METHOD findSearchResults
VAR_INPUT
END_VAR
VAR
	i : INT;
	j : INT;
	searchResult : ST_SearchResult;
END_VAR
FOR i:=0 TO stDoorTrack.CandidateRoutes.CandidateRoutesCount - 1 DO
	FOR j:=0 TO stDoorTrack.CandidateRoutes.CandidateRoutes[i].PathsInfoCount - 1 DO
		searchResult := stSearchResultDefault;
		searchResult.PathIno := stDoorTrack.CandidateRoutes.CandidateRoutes[i].PathsInfo[j];
		searchResult.TargetFeedoutSide := stDoorTrack.CandidateRoutes.CandidateRoutes[i].TargetFeedoutSide;
		addSearchResultToDoorTrack(searchResult);
	END_FOR
END_FOR
END_METHOD

METHOD getFeedMgrStateDescription : STRING
IF config_bIsConveyorTable THEN
	getFeedMgrStateDescription := smC235FeedManager.getStateDescription();
ELSE
	getFeedMgrStateDescription := smC234FeedManager.getStateDescription();
END_IF
END_METHOD

METHOD getSourceAndDestinationIndexFeedoutPortsCount : UINT
IF stDoorTrack.Source < 0 OR stDoorTrack.Source >= MAX_TABLES_COUNT OR
	stDoorTrack.DestinationIndex < 0 OR stDoorTrack.DestinationIndex >= MAX_FEEDOUT_PORTS THEN
	getSourceAndDestinationIndexFeedoutPortsCount := 0;
	RETURN;
END_IF
getSourceAndDestinationIndexFeedoutPortsCount := 
	MAIN.mainStateMachine.smCtrlInterface.
		config_stTransferTableConfig.PrimaryTable.
		Tables[stDoorTrack.Source].DestinationsFeedoutPortsMappingConfig.
		DestinationsFeedoutPortsMappings[stDoorTrack.DestinationIndex].FeedoutPortsCount;
END_METHOD

METHOD getStateDescription : STRING
CASE machineState OF

	TABLEMANAGER_DISABLED:
		getStateDescription := 'Disabled';
			
	TABLEMANAGER_ENABLING:
		getStateDescription := 'Enabling';
			
	TABLEMANAGER_INLINE_JOGGING:
		getStateDescription := 'Inline Jogging';
			
	TABLEMANAGER_CROSS_JOGGING:
		getStateDescription := 'Cross Jogging';
		
	TABLEMANAGER_TO_FENCE_JOGGING:
		getStateDescription := 'To-Fence Jogging';
	
	TABLEMANAGER_ROTATE:
		getStateDescription := 'Rotating';
			
	TABLEMANAGER_SELF_CENTER:
		getStateDescription := 'Centering';
			
	TABLEMANAGER_AUTOFEED_OFF:
		getStateDescription := 'Autofeed Off';
			
	TABLEMANAGER_AUTOFEED_ON:
		getStateDescription := 'Autofeed On';
		
	TABLEMANAGER_DOOR_TRACKER_START:
		getStateDescription := 'Door Track Starting';
			
	TABLEMANAGER_DOOR_TRACKER_WAIT_FOR_DATA_READY_OR_TRANSFERRED_IN:
		IF config_bCanFeedinFromSideA THEN
			getStateDescription := 'Waiting for Door Data Ready or Transferred In';
		ELSE
			getStateDescription := 'Waiting for Door Transferred In';
		END_IF
		
	TABLEMANAGER_DOOR_TRACKER_TRANSFERRING_IN:
		getStateDescription := 'Transferring In';
			
	TABLEMANAGER_DOOR_TRACKER_ROUTE_READY_WAIT_FOR_FEED_IN:
		getStateDescription := 'Route Ready - Waiting for Feed In';
			
	TABLEMANAGER_DOOR_TRACKER_DOOR_FEEDING_IN:
		getStateDescription := 'Door Feeding In';
		
	TABLEMANAGER_DOOR_TRACKER_DOOR_IN_MACHINE_IDLE:
		getStateDescription := 'Door in Machine - Waiting for Transferred Out';

	TABLEMANAGER_DOOR_TRACKER_WAIT_FOR_FEED_OUT:
		IF cmd_bDoorDataReadyLatched THEN
			getStateDescription := 'Waiting for Feed Out. Data Ready Latch Active';
		ELSE
			getStateDescription := 'Waiting for Feed Out';
		END_IF
		
			
	TABLEMANAGER_DOOR_TRACKER_DOOR_FEEDING_OUT:
		getStateDescription := 'Feeding Out';
		
	TABLEMANAGER_DOOR_TRACKER_WAIT_ALL_TABLES_READY:
		getStateDescription := 'Waiting for All Tables Ready';
		
	TABLEMANAGER_DOOR_TRACKER_TRANSFERRING_OUT:
		getStateDescription := 'Transferring Out';
			
	TABLEMANAGER_DOOR_TRACKER_COMPLETE:
		getStateDescription := 'Completed';			
		
	TABLEMANAGER_DOOR_TRACKER_FINDPATH_INIT:
		getStateDescription := 'Finding Path Init';
	
	TABLEMANAGER_DOOR_TRACKER_FINDPATH_RESET:
		getStateDescription := 'Resetting Door Tracker';
		
	TABLEMANAGER_DOOR_TRACKER_FINDPATH_FIND_ENABLED_FEEDOUT_PORTS:
		getStateDescription := 'Finding Enabled Feedout Ports';
		
	TABLEMANAGER_DOOR_TRACKER_FINDPATH_WAITING_FOR_CLEAR_ROUTE:
		getStateDescription := 'Waiting for Clear Route';
	
	TABLEMANAGER_DOOR_TRACKER_FINDPATH_FIND_CANDIDATE_ROUTES:
		getStateDescription := 'Finding Candidate Routes';
		
	TABLEMANAGER_DOOR_TRACKER_FINDPATH_FIND_SEARCH_RESULTS:
		getStateDescription := 'Finding Search Results';
		
	TABLEMANAGER_DOOR_TRACKER_FINDPATH_COMPUTE_FINAL_SCORE:
		getStateDescription := 'Computing Final Score';
		
	TABLEMANAGER_DOOR_TRACKER_FINDPATH_REQUEST_NEW_ROUTE_COMPLETE:
		getStateDescription := 'Request New Route Complete';
		
	TABLEMANAGER_DOOR_TRACKER_FINDPATH_COMPLETE:
		getStateDescription := 'Finding Path Complete';
	
	TABLEMANAGER_DOOR_TRACKER_ALL_TARGET_FEEDOUT_PORTS_DISABLED:
		getStateDescription := 'All of Target Feed-out Ports Disabled';	

	TABLEMANAGER_DOOR_TRACKER_DOOR_HAS_NO_TARGET:
		getStateDescription := 'Door Has No Target';
		
	TABLEMANAGER_ERROR:
		getStateDescription := 'Error';
		
END_CASE
END_METHOD

METHOD getTargetNodeDirection : E_Direction
VAR 
	i : INT;
END_VAR
getTargetNodeDirection := E_Direction.None;
IF NOT bHasDoor THEN
	RETURN;
END_IF

FOR i:= 0 TO stDoorTrack.TargetPath.PathCount - 1 DO
	// do we have the source from TargetPath?
	IF stDoorTrack.TargetPath.Path[i].TableIndex = config_iTableArrayIndex THEN
		getTargetNodeDirection := stDoorTrack.TargetPath.Path[i].Direction;
		RETURN;
	END_IF
END_FOR
END_METHOD

METHOD goFast
VAR_INPUT
END_VAR
psmHcFeedMotor^.cmd_bSpeedFast := TRUE;
END_METHOD

METHOD goFwd
VAR_INPUT
END_VAR
psmHcFeedMotor^.cmd_bFwd := TRUE;
END_METHOD

METHOD goRev
VAR_INPUT
END_VAR
psmHcFeedMotor^.cmd_bRev := TRUE;
END_METHOD

METHOD goSlow
VAR_INPUT
END_VAR
psmHcFeedMotor^.cmd_bSpeedSlow := TRUE;
END_METHOD

METHOD hasDeadlockedDoorInPath : BOOL
VAR_INPUT
	pstPath : POINTER TO ST_PathInfo;
END_VAR
VAR
	i : INT;
END_VAR
hasDeadlockedDoorInPath := FALSE;
IF pstPath = 0 THEN	
	RETURN;
END_IF

FOR i:= 0 TO pstPath^.PathCount - 1 DO
	IF MAIN.mainStateMachine.asmTableManagers[pstPath^.Path[i].TableIndex].bHasDoor AND 
		(MAIN.mainStateMachine.asmTableManagers[pstPath^.Path[i].TableIndex].bWaitingForClearRoute OR
		MAIN.mainStateMachine.asmTableManagers[pstPath^.Path[i].TableIndex].bAllTargetFeedoutPortsDisabled OR
		MAIN.mainStateMachine.asmTableManagers[pstPath^.Path[i].TableIndex].bDoorHasNoTarget)
	THEN
		hasDeadlockedDoorInPath := TRUE;
		RETURN;
	END_IF
END_FOR
END_METHOD

METHOD hasDoorGoingOppositeDirection : BOOL
VAR_INPUT
	pstPath : POINTER TO ST_PathInfo;
END_VAR
VAR
	i : INT;
	j : INT;
	k : INT;
	intersectAtTableIndex : INT;
	prevDoorDirection : E_Direction;
	curDoorDirection : E_Direction;
	otherDoorDirection : E_Direction;
	pstPathOther : POINTER TO ST_PathInfo;
END_VAR
hasDoorGoingOppositeDirection := FALSE;
IF pstPath = 0 THEN	
	RETURN;
END_IF

FOR i:= 0 TO pstPath^.PathCount - 1 DO
	intersectAtTableIndex := pstPath^.Path[i].TableIndex;
	IF MAIN.mainStateMachine.asmTableManagers[intersectAtTableIndex].stDoorTrack.Target <> -1 THEN
		pstPathOther := ADR(MAIN.mainStateMachine.asmTableManagers[intersectAtTableIndex].stDoorTrack.TargetPath);
		FOR j:= 0 TO pstPathOther^.PathCount - 1 DO
			prevDoorDirection := E_Direction.None;
			FOR k:= 0 TO pstPath^.PathCount - 1 DO				
				curDoorDirection := pstPath^.Path[k].Direction;
				IF pstPathOther^.Path[j].TableIndex = pstPath^.Path[k].TableIndex THEN
					otherDoorDirection  := pstPathOther^.Path[j].Direction;
					IF 	curDoorDirection = E_Direction.North 	AND otherDoorDirection = E_Direction.South OR
						curDoorDirection = E_Direction.South 	AND otherDoorDirection = E_Direction.North OR
						curDoorDirection = E_Direction.West 	AND otherDoorDirection = E_Direction.East OR
						curDoorDirection = E_Direction.East 	AND otherDoorDirection = E_Direction.West OR
						prevDoorDirection = E_Direction.North 	AND otherDoorDirection = E_Direction.South OR
						prevDoorDirection = E_Direction.South 	AND otherDoorDirection = E_Direction.North OR
						prevDoorDirection = E_Direction.West 	AND otherDoorDirection = E_Direction.East OR
						prevDoorDirection = E_Direction.East 	AND otherDoorDirection = E_Direction.West
					THEN
						hasDoorGoingOppositeDirection := TRUE;
						RETURN;
					END_IF
				END_IF
				prevDoorDirection := curDoorDirection;
			END_FOR
		END_FOR
	END_IF
END_FOR
END_METHOD

METHOD hasEmptyTableInPath : BOOL
VAR_INPUT
	pstPath : POINTER TO ST_PathInfo;
END_VAR
VAR
	i : INT;
END_VAR
IF pstPath = 0 THEN
	hasEmptyTableInPath := FALSE;
	RETURN;
END_IF

IF pstPath^.PathCount = 0 THEN
	hasEmptyTableInPath := FALSE;
	RETURN;
END_IF

IF pstPath^.PathCount = 1 THEN
	hasEmptyTableInPath := NOT MAIN.mainStateMachine.asmTableManagers[pstPath^.Path[0].TableIndex].bHasDoor;
	RETURN;
END_IF

// skip index 0, which is the source/first table in path.
FOR i:= 1 TO pstPath^.PathCount - 1 DO
	IF NOT MAIN.mainStateMachine.asmTableManagers[pstPath^.Path[i].TableIndex].bHasDoor THEN
		hasEmptyTableInPath := TRUE;
		RETURN;
	END_IF
END_FOR

hasEmptyTableInPath := FALSE;
END_METHOD

METHOD hasError : bool
hasError := smDoorDasher.bError;
IF hasError THEN
	RETURN;
END_IF

IF config_bIsConveyorTable THEN
	hasError := smC235FeedManager.bError;
ELSE
	hasError := smC234FeedManager.bError;
END_IF
END_METHOD

METHOD hasErrorDescription : T_MaxString
hasErrorDescription := smDoorDasher.sError;
IF hasErrorDescription <> '' THEN
	RETURN;
END_IF

IF config_bIsConveyorTable THEN
	hasErrorDescription := smC235FeedManager.sError;
ELSE
	hasErrorDescription := smC234FeedManager.sError;
END_IF
END_METHOD

METHOD hasErrorId : UINT
hasErrorId := INT_TO_UINT(smDoorDasher.iLastErrorId);
IF hasErrorId <> 0 THEN
	RETURN;
END_IF

IF config_bIsConveyorTable THEN
	hasErrorId := INT_TO_UINT(smC235FeedManager.iLastErrorId);
ELSE
	hasErrorId := INT_TO_UINT(smC234FeedManager.iLastErrorId);
END_IF
END_METHOD

METHOD hasIncomingDoorInPath : BOOL
VAR_INPUT
	pstPath : POINTER TO ST_PathInfo;
END_VAR
VAR
	i : INT;
END_VAR
hasIncomingDoorInPath := FALSE;
IF pstPath = 0 THEN	
	RETURN;
END_IF

FOR i:= 0 TO pstPath^.PathCount - 1 DO
	IF MAIN.mainStateMachine.asmTableManagers[pstPath^.Path[i].TableIndex].bRouteReadyWaitForFeedIn THEN
		hasIncomingDoorInPath := TRUE;
		RETURN;
	END_IF
END_FOR
END_METHOD

METHOD initDoorTrack
VAR_INPUT
END_VAR
stDoorTrackLast := stDoorTrack; 

stDoorTrack.CandidateRoutes := stCandidateRoutesDefault;
stDoorTrack.SearchResults := stSearchResultsDefault;
stDoorTrack.TargetPath := stPathInfoDefault;

bHasEnabledFeedoutPorts := FALSE;

IF cmd_bRequestNewRoute THEN
	stDoorTrack.AllEnabledFeedoutPorts := stFeedoutPortsConfigDefault;
	stDoorTrack.RejectedFeedoutPorts := stFeedoutPortsConfigDefault;
	stDoorTrack.ReroutableFeedoutPorts := stReroutableFeedoutPortsConfigDefault;
	stDoorTrack.RejectedFeedoutPorts.FeedoutPortsCount := -1; // Notifies HMI to clear the rejected feed-out ports list for operator's manual re-route.
	stDoorTrack.ReroutableFeedoutPorts.FeedoutPortsCount := -1; // Notifies HMI to clear the reroutable feed-out ports list for operator's manual re-route.
ELSE
	stDoorTrack.TargetFeedoutPorts := stFeedoutPortsConfigDefault;
	stDoorTrack.DoorIsRotating := FALSE;
	stDoorTrack.DoorRotateRequired := FALSE;
	stDoorTrack.DoorWasRotated := FALSE;
END_IF
END_METHOD

METHOD initialize
VAR CONSTANT		
END_VAR
SUPER^.initialize();

descriptor.sModuleClass := 'TableManager';

// TODO: don't init if config_pstHcTransferTableHardware and config_pstHcConveyorHardware are null
config_pstHcTransferTableHardware;
config_pstHcConveyorHardware;

// initialize machine configs and defaults
cmd_bManualControlEnabled := config_bManualControlEnabled;

(*     --- Feed System ---     *)
IF config_bIsConveyorTable THEN
	//
	iCrossFeedFastSpeedRpm	:= LREAL_TO_UINT(config_iCrossFeedFastSpeedFPM / CONVEYOR_CROSSFEED_RPM_TO_FPM);
	iCrossFeedSlowSpeedRpm	:= LREAL_TO_UINT(config_iCrossFeedSlowSpeedFPM / CONVEYOR_CROSSFEED_RPM_TO_FPM);
	iFeedFastSpeedRPM		:= iCrossFeedFastSpeedRpm;
	iFeedSlowSpeedRPM 		:= iCrossFeedSlowSpeedRpm;
	iFeedOutSpeedRPM		:= 0; // not used for Conveyor table
	IF (config_pstHcConveyorHardware <> 0) THEN
		psmHcFeedMotor := ADR(config_pstHcConveyorHardware^.smFeedMotor);
	END_IF
ELSE
	//
	iCrossFeedFastSpeedRpm	:= LREAL_TO_UINT(config_iCrossFeedFastSpeedFPM / TABLE_CROSSFEED_RPM_TO_FPM);
	iCrossFeedSlowSpeedRpm	:= LREAL_TO_UINT(config_iCrossFeedSlowSpeedFPM / TABLE_CROSSFEED_RPM_TO_FPM);
	iFeedFastSpeedRPM		:= LREAL_TO_UINT(config_iFeedFastSpeedFPM / TABLE_INLINE_FEED_RPM_TO_FPM);
	iFeedSlowSpeedRPM 		:= LREAL_TO_UINT(config_iFeedSlowSpeedFPM / TABLE_INLINE_FEED_RPM_TO_FPM);
	iFeedOutSpeedRPM		:= LREAL_TO_UINT(config_iFeedOutSpeedFPM  / TABLE_INLINE_FEED_RPM_TO_FPM);
	IF (config_pstHcTransferTableHardware <> 0) THEN
		psmHcFeedMotor := ADR(config_pstHcTransferTableHardware^.smFeedMotor);
	END_IF
END_IF

IF (psmHcFeedMotor = 0) THEN
	logger(ePriority := E_LogPriority.LOGPRIORITY_WARNING_LOW, sMessage := 'Incorrect config - assigning dummy pointer to VFD');
	psmHcFeedMotor := ADR(MAIN.mainStateMachine.smDummyMotor);
END_IF
	
{IF defined (noHW) OR defined (noHW_UML)}
	// these are for no hardware mode only...
	psmHcFeedMotor^.config_bNoHardwareTestMode := config_bNoHardwareTestMode;
	psmHcFeedMotor^.config_fTestMaxAccel := 24; // unit: in/s^2
	psmHcFeedMotor^.config_fTestMaxDecel := 24; // unit: in/s^2
	psmHcFeedMotor^.config_fTestMaxJerk := 144; // unit: in/s^3
	psmHcFeedMotor^.config_fTestMaxSpeed := 30; // unit : in/sec
	
	IF psmHcFeedMotor^.config_iFastSpeedRPM = 0 THEN
		psmHcFeedMotor^.config_iFastSpeedRPM := 1345;
	END_IF
	psmHcFeedMotor^.config_fUnitConversionFactor := (config_iFeedFastSpeedFPM * 12.0) / (psmHcFeedMotor^.config_iFastSpeedRPM * 60.0);
{END_IF}

// Assign dummy values preemptively - if have correct link to hardware, will get overwritten
// Have to assign these here, in initialize, because SM_TableManager references some of these in preProcess
smC234FeedManager.psmCrossFeedFenceHeightCyl 					:= ADR(MAIN.mainStateMachine.smDummyCylinder);
smC234FeedManager.psmCrossFeedTransferHeightCyl 				:= ADR(MAIN.mainStateMachine.smDummyCylinder);
smC234FeedManager.smSelfCenterManager.psmSelfCenterWheelsCyl 	:= ADR(MAIN.mainStateMachine.smDummyCylinder);
smC234FeedManager.smSelfCenterManager.psmSelfCenterCyl 			:= ADR(MAIN.mainStateMachine.smDummyCylinder);
smC234FeedManager.smRotateManager.psmDoorLiftCyl				:= ADR(MAIN.mainStateMachine.smDummyCylinder);
smC234FeedManager.smRotateManager.psmRotateCyl					:= ADR(MAIN.mainStateMachine.smDummyDoubleCylinder);
	
IF config_bIsConveyorTable THEN
	addChildStateMachine('C235 Feed Manager', ADR(smC235FeedManager)); 
		smC235FeedManager.pbTableIsEmpty := ADR(bTableIsEmpty);
		smC235FeedManager.pbDoorInMachine := ADR(bDoorInMachine);
		smC235FeedManager.pstTable := THIS;
		smC235FeedManager.pstDoorTrack := ADR(stDoorTrack);
		smC235FeedManager.itfDoorTracker := THIS^;
		smC235FeedManager.psmFeedMotor := psmHcFeedMotor;
		smC235FeedManager.config_iFeedOutSpeedRPM := iCrossFeedFastSpeedRPM;
		smC235FeedManager.config_iCrossFastSpeedRPM := iCrossFeedFastSpeedRPM;
		smC235FeedManager.config_iCrossSlowSpeedRPM := iCrossFeedSlowSpeedRPM;
		smC235FeedManager.config_bNoHardwareTestMode := config_bNoHardwareTestMode;
		smC235FeedManager.config_iTableArrayIndex := config_iTableArrayIndex;
ELSE		
	addChildStateMachine('C234 Feed Manager', ADR(smC234FeedManager));
		smC234FeedManager.pbTableIsEmpty := ADR(bTableIsEmpty);
		smC234FeedManager.pbDoorInMachine := ADR(bDoorInMachine);
		smC234FeedManager.pstTable := THIS;
		smC234FeedManager.pstDoorTrack := ADR(stDoorTrack);
		smC234FeedManager.itfDoorTracker := THIS^;
		smC234FeedManager.config_bCanRotate := config_bCanRotate;
		smC234FeedManager.config_bCanSelfCenter := config_bCanSelfCenter;
		smC234FeedManager.config_bIsBufferTable := config_bIsBufferTable;
		smC234FeedManager.psmFeedMotor := psmHcFeedMotor;
		smC234FeedManager.config_iFastSpeedRPM := iFeedFastSpeedRPM;
		smC234FeedManager.config_iSlowSpeedRPM := iFeedSlowSpeedRPM;
		smC234FeedManager.config_iFeedOutSpeedRPM := iFeedOutSpeedRPM;
		smC234FeedManager.config_iCrossFastSpeedRPM := iCrossFeedFastSpeedRPM;
		smC234FeedManager.config_iCrossSlowSpeedRPM := iCrossFeedSlowSpeedRPM;
		smC234FeedManager.config_bNoHardwareTestMode := config_bNoHardwareTestMode;
		smC234FeedManager.config_iTableArrayIndex := config_iTableArrayIndex;
		// Assign valve pointers
		IF (config_pstHcTransferTableHardware <> 0) THEN
			smC234FeedManager.psmCrossFeedFenceHeightCyl 					:= ADR(config_pstHcTransferTableHardware^.smCrossFeedFenceHeightCyl);
			smC234FeedManager.psmCrossFeedTransferHeightCyl 				:= ADR(config_pstHcTransferTableHardware^.smCrossFeedTransferHeightCyl);
			smC234FeedManager.smSelfCenterManager.psmSelfCenterWheelsCyl 	:= ADR(config_pstHcTransferTableHardware^.smSelfCenterWheelsCyl);
			smC234FeedManager.smSelfCenterManager.psmSelfCenterCyl 			:= ADR(config_pstHcTransferTableHardware^.smSelfCenterCyl);
			smC234FeedManager.smRotateManager.psmDoorLiftCyl 				:= ADR(config_pstHcTransferTableHardware^.smDoorLiftCyl);
			smC234FeedManager.smRotateManager.psmRotateCyl 					:= ADR(config_pstHcTransferTableHardware^.smRotateCyl);
		ELSE
			logger(ePriority := E_LogPriority.LOGPRIORITY_WARNING_LOW, sMessage := 'Incorrect config - assigning dummy pointer to valves');
		END_IF
END_IF

addChildStateMachine('Door Dasher', ADR(smDoorDasher));
	smDoorDasher(
		pstTable := THIS,
		pstDoorTrack := ADR(stDoorTrack),
		itfDoorTracker := THIS^,
		config_bNoHardwareTestMode := config_bNoHardwareTestMode,
		config_iTableArrayIndex := config_iTableArrayIndex
	);
END_METHOD

METHOD initInputSourceAndDestinationIndexWithHighestFeedoutPortsCount : BOOL
VAR_IN_OUT
	iInputSource	: INT;
	iDestinationIndex	: INT;
END_VAR
VAR 
	iInputSourceIndex : INT;
	iDestIndex : INT;
	feedoutPortsCountMax : INT;
END_VAR
iInputSource := 0;
iDestinationIndex := 0;
feedoutPortsCountMax := 0;

FOR iInputSourceIndex:=0 TO MAIN.mainStateMachine.smCtrlInterface.config_stTransferTableConfig.PrimaryTable.TablesCount-1 DO
	IF NOT (MAIN.mainStateMachine.smCtrlInterface.config_stTransferTableConfig.PrimaryTable.Tables[iInputSourceIndex].IsFunctionalTable AND
			MAIN.mainStateMachine.asmTableManagers[iInputSourceIndex].config_bCanFeedinFromSideA) THEN
		CONTINUE;
	END_IF
	IF MAIN.mainStateMachine.smCtrlInterface.config_stTransferTableConfig.PrimaryTable.Tables[iInputSourceIndex].DestinationsFeedoutPortsMappingConfig.DestinationsFeedoutPortsMappingsCount > 0 THEN
		FOR iDestIndex:=0 TO MAIN.mainStateMachine.smCtrlInterface.config_stTransferTableConfig.PrimaryTable.Tables[iInputSourceIndex].DestinationsFeedoutPortsMappingConfig.DestinationsFeedoutPortsMappingsCount - 1 DO
			IF MAIN.mainStateMachine.smCtrlInterface.config_stTransferTableConfig.PrimaryTable.Tables[iInputSourceIndex].DestinationsFeedoutPortsMappingConfig.DestinationsFeedoutPortsMappings[iDestIndex].FeedoutPortsCount > feedoutPortsCountMax THEN
				iInputSource := iInputSourceIndex;
				iDestinationIndex := MAIN.mainStateMachine.smCtrlInterface.config_stTransferTableConfig.PrimaryTable.Tables[iInputSourceIndex].DestinationsFeedoutPortsMappingConfig.DestinationsFeedoutPortsMappings[iDestIndex].DestinationIndex;
				feedoutPortsCountMax := MAIN.mainStateMachine.smCtrlInterface.config_stTransferTableConfig.PrimaryTable.Tables[iInputSourceIndex].DestinationsFeedoutPortsMappingConfig.DestinationsFeedoutPortsMappings[iDestIndex].FeedoutPortsCount;
			END_IF
		END_FOR
	END_IF
END_FOR
END_METHOD

METHOD isCurrentTargetFeedoutPortEnabled : BOOL
VAR_INPUT
END_VAR
isCurrentTargetFeedoutPortEnabled := FALSE;
IF 	stDoorTrack.Target <> -1 THEN		
	isCurrentTargetFeedoutPortEnabled := MAIN.mainStateMachine.asmTableManagers[stDoorTrack.Target].isFeedoutSideEnabled(stDoorTrack.TargetFeedoutSide);
END_IF
END_METHOD

// if currentTargetFeedoutPort exists in DestinationIndex, then the current Target was a re-route.
METHOD isCurrentTargetFeedoutPortExistInDestinationIndexFeedoutPorts : BOOL
VAR_INPUT
END_VAR
VAR
	i : INT;
	j : INT;
	k : INT;
	stFeedoutPort : ST_FeedoutPort;
END_VAR
isCurrentTargetFeedoutPortExistInDestinationIndexFeedoutPorts := FALSE;
IF 	stDoorTrack.DestinationIndex <> -1 AND
	stDoorTrack.Target <> -1 
	THEN
	i := stDoorTrack.Source;
	IF MAIN.mainStateMachine.smCtrlInterface.config_stTransferTableConfig.PrimaryTable.Tables[i].DestinationsFeedoutPortsMappingConfig.DestinationsFeedoutPortsMappingsCount > 0 THEN
		FOR j:=0 TO MAIN.mainStateMachine.smCtrlInterface.config_stTransferTableConfig.PrimaryTable.Tables[i].DestinationsFeedoutPortsMappingConfig.DestinationsFeedoutPortsMappingsCount - 1 DO
			IF MAIN.mainStateMachine.smCtrlInterface.config_stTransferTableConfig.PrimaryTable.Tables[i].DestinationsFeedoutPortsMappingConfig.DestinationsFeedoutPortsMappings[j].DestinationIndex = stDoorTrack.DestinationIndex THEN
				IF MAIN.mainStateMachine.smCtrlInterface.config_stTransferTableConfig.PrimaryTable.Tables[i].DestinationsFeedoutPortsMappingConfig.DestinationsFeedoutPortsMappings[j].FeedoutPortsCount > 0 THEN
					FOR k:=0 TO MAIN.mainStateMachine.smCtrlInterface.config_stTransferTableConfig.PrimaryTable.Tables[i].DestinationsFeedoutPortsMappingConfig.DestinationsFeedoutPortsMappings[j].FeedoutPortsCount - 1 DO
						stFeedoutPort := MAIN.mainStateMachine.smCtrlInterface.config_stTransferTableConfig.PrimaryTable.Tables[i].DestinationsFeedoutPortsMappingConfig.DestinationsFeedoutPortsMappings[j].FeedoutPorts[k];
						IF stFeedoutPort.TableIndex = stDoorTrack.Target AND stFeedoutPort.Side = stDoorTrack.TargetFeedoutSide THEN
							isCurrentTargetFeedoutPortExistInDestinationIndexFeedoutPorts := TRUE;
							RETURN;
						END_IF
					END_FOR
				END_IF
				EXIT;
			END_IF
		END_FOR
	END_IF
END_IF
END_METHOD

METHOD isFeedoutSideEnabled : BOOL
VAR_INPUT
	eFeedoutSide : E_FeedoutSideType;
END_VAR
isFeedoutSideEnabled := FALSE;
IF config_bIsConveyorTable THEN
	IF eFeedoutSide = E_FeedoutSideType.C THEN
		isFeedoutSideEnabled := NOT smC235FeedManager.di_DisableFeedoutSideC;
	ELSIF eFeedoutSide = E_FeedoutSideType.D THEN
		isFeedoutSideEnabled := NOT smC235FeedManager.di_DisableFeedoutSideD;
	END_IF
ELSE
	IF eFeedoutSide = E_FeedoutSideType.A THEN
		isFeedoutSideEnabled := NOT smC234FeedManager.di_DisableFeedoutSideA;
	ELSIF eFeedoutSide = E_FeedoutSideType.B THEN
		isFeedoutSideEnabled := NOT smC234FeedManager.di_DisableFeedoutSideB;
	ELSIF eFeedoutSide = E_FeedoutSideType.C THEN
		isFeedoutSideEnabled := NOT smC234FeedManager.di_DisableFeedoutSideC;
	ELSIF eFeedoutSide = E_FeedoutSideType.D THEN
		isFeedoutSideEnabled := NOT smC234FeedManager.di_DisableFeedoutSideD;
	END_IF
END_IF
END_METHOD

METHOD isNeighborInTargetPath : BOOL
VAR_INPUT
	neighborIndex : INT;
END_VAR
VAR 
	i : INT;
END_VAR
isNeighborInTargetPath := FALSE;

FOR i:= 0 TO stDoorTrack.TargetPath.PathCount - 1 DO
	// do we have the neighborIndex in TargetPath?
	IF stDoorTrack.TargetPath.Path[i].TableIndex = neighborIndex THEN
		isNeighborInTargetPath := TRUE;
		RETURN;
	END_IF
END_FOR
END_METHOD

METHOD isTableIndexExistInCandidateRoutes : BOOL
VAR_INPUT
	iTableIndex : INT;
END_VAR
VAR
	i : INT;
END_VAR
isTableIndexExistInCandidateRoutes := FALSE;
FOR i:=0 TO stDoorTrack.CandidateRoutes.CandidateRoutesCount-1 DO
	IF stDoorTrack.CandidateRoutes.CandidateRoutes[i].TargetTableIndex = iTableIndex THEN
		isTableIndexExistInCandidateRoutes := TRUE;
		RETURN;
	END_IF
END_FOR
END_METHOD

METHOD minDirectionalChanges : LREAL
VAR_INPUT
	pstSearchResults : POINTER TO ST_SearchResults;
END_VAR
VAR
	i : INT;
	pstSearchResult : POINTER TO ST_SearchResult;
	minDirChanges : LREAL := MAX_LREAL;
END_VAR
IF pstSearchResults = 0 THEN
	RETURN;
END_IF

FOR i:=0 TO pstSearchResults^.SearchResultsCount - 1 DO
	pstSearchResult := ADR(pstSearchResults^.SearchResults[i]);
	IF pstSearchResult^.DirectionalChanges < minDirChanges THEN
		minDirChanges := pstSearchResult^.DirectionalChanges;
	END_IF
END_FOR

minDirectionalChanges := minDirChanges;
END_METHOD

METHOD minDoorsInPath : LREAL
VAR_INPUT
	pstSearchResults : POINTER TO ST_SearchResults;
END_VAR
VAR
	i : INT;
	pstSearchResult : POINTER TO ST_SearchResult;
	minDoorIntersects : LREAL := MAX_LREAL;
END_VAR
IF pstSearchResults = 0 THEN
	RETURN;
END_IF

FOR i:=0 TO pstSearchResults^.SearchResultsCount - 1 DO
	pstSearchResult := ADR(pstSearchResults^.SearchResults[i]);
	IF pstSearchResult^.DoorsInPath < minDoorIntersects THEN
		minDoorIntersects := pstSearchResult^.DoorsInPath;
	END_IF
END_FOR

minDoorsInPath := minDoorIntersects;
END_METHOD

METHOD minNumberOfHops : LREAL
VAR_INPUT
	pstSearchResults : POINTER TO ST_SearchResults;
END_VAR
VAR
	i : INT;
	pstSearchResult : POINTER TO ST_SearchResult;
	minHops : LREAL := MAX_LREAL;
END_VAR
IF pstSearchResults = 0 THEN
	RETURN;
END_IF

FOR i:=0 TO pstSearchResults^.SearchResultsCount - 1 DO
	pstSearchResult := ADR(pstSearchResults^.SearchResults[i]);
	IF pstSearchResult^.NumberOfHops < minHops THEN
		minHops := pstSearchResult^.NumberOfHops;
	END_IF
END_FOR

minNumberOfHops := minHops;
END_METHOD

METHOD pathHasRotateOption : BOOL
VAR_INPUT
	pstPath : POINTER TO ST_PathInfo;
END_VAR
VAR
	i : INT;
	nodeTableIndex : INT;
END_VAR
pathHasRotateOption := FALSE;
IF pstPath = 0 THEN	
	RETURN;
END_IF

FOR i:= 0 TO pstPath^.PathCount - 1 DO
	nodeTableIndex := pstPath^.Path[i].TableIndex;
	IF MAIN.mainStateMachine.asmTableManagers[nodeTableIndex].config_bCanRotate THEN
		pathHasRotateOption := TRUE;
		RETURN;
	END_IF
END_FOR
END_METHOD

METHOD postProcess
VAR_INPUT
END_VAR
SUPER^.postProcess();
cmd_bAbort := FALSE;
cmd_bRotate			:= FALSE;
cmd_bSelfCenter			:= FALSE;	
cmd_bExternal		:= FALSE;	
cmd_bInternal			:= FALSE;	
cmd_bFeedinStarted	:= FALSE;
cmd_bFeedinCompleted := FALSE;
cmd_bFeedoutStarted := FALSE;
cmd_bFeedoutCompleted := FALSE;
cmd_bDoorTransferInStarted := FALSE;
cmd_bDoorTransferInCompleted := FALSE;
cmd_bDoorTransferOutCompleted := FALSE;
END_METHOD

(* this method is run before the doState is run*)
METHOD preProcess
SUPER^.preProcess();

// Jamb kickover
IF (config_pstHcTransferTableHardware <> 0) THEN
	tofJambKickOverTimer(IN:=config_bCanFeedinFromSideA AND config_pstHcTransferTableHardware^.di_JambKickoverEye, PT:=T#2.0S);
	config_pstHcTransferTableHardware^.do_jambKickover := tofJambKickOverTimer.Q AND (NOT config_pstHcTransferTableHardware^.di_JambKickoverEye);
END_IF

// persist configs to disk
rtrigPersistentDataChanged(CLK:=
	config_bManualControlEnabled <> cmd_bManualControlEnabled);
IF rtrigPersistentDataChanged.Q THEN
	config_bManualControlEnabled := cmd_bManualControlEnabled;
END_IF
bExternal := anyChildExternal();
status_bBusy := anyChildBusy() OR smDoorDasher.status_bBusy;
status_bMoving := psmHcFeedMotor^.status_bMoving;
bReadyToRotate := 
	NOT (smC234FeedManager.smRotateManager.psmDoorLiftCyl^.status_bFloating OR smC234FeedManager.smRotateManager.psmRotateCyl^.status_bFloating) AND
	(smC234FeedManager.smSelfCenterManager.psmSelfCenterCyl^.status_bRetracted OR NOT config_bCanSelfCenter);
bOkToSelfCenter := smC234FeedManager.smRotateManager.bDoorLiftCylRetracted OR NOT config_bCanRotate;

bHasDoor := bDoorInMachine;
ftrigHasDoor(CLK:=bHasDoor);

rtrigAutofeedOn(CLK:=cmd_bAutoFeedOn);
IF rtrigAutofeedOn.Q THEN
	autofeedOn();
END_IF

// Eye blowoff
IF (config_pstHcTransferTableHardware <> 0) THEN
	IF rtrigAutofeedOn.Q OR ftrigHasDoor.Q THEN
		config_pstHcTransferTableHardware^.do_eyeBlowoff := TRUE;
	END_IF
	tonEyeBlowoffTimer(IN:=config_pstHcTransferTableHardware^.do_eyeBlowoff, PT:=T#1S);
	IF tonEyeBlowoffTimer.Q THEN
		config_pstHcTransferTableHardware^.do_eyeBlowoff := FALSE;
	END_IF
END_IF

ftrigAnyChildNotAutofeedOn(CLK:=allChildrenAutoFeedOn());
IF ftrigAnyChildNotAutofeedOn.Q THEN
	cmd_bAutoFeedOn := FALSE;
END_IF

ftrigAutofeedOn(CLK:=cmd_bAutoFeedOn);
IF ftrigAutofeedOn.Q THEN
	autofeedOff();
END_IF


rtrigExternal(CLK:=cmd_bExternal);
IF rtrigExternal.Q THEN
	setExternal();
END_IF

rtrigExternal(CLK:=cmd_bInternal);
IF rtrigExternal.Q THEN
	setInternal();
END_IF

rtrigTableIndexNotExistInDoorTrackTargetPath(CLK:= 
	bHasDoor AND 
	stDoorTrack.Target <> -1 AND 
	stDoorTrack.TargetPath.PathCount > 0 AND 
	NOT existTableIndexInDoorTrackTargetPath());

rtrigRequestNewRoute(CLK:=cmd_bRequestNewRoute);

// cmd_bIncomingDoorHandValid := di_IncomingDoorLH XOR di_IncomingDoorRH
cmd_bIncomingDoorHandValid := cmd_eIncomingDoorHand <> E_DOORHAND.DOORHAND_NO_HAND;

// Monitor cmd_bIncomingDoorHandValid on falling edge. The feeding machine (ie, 994-X) clears LH/RH inputs on completion of its feed-out seq. 
ftrigIncomingDoorHandValid(CLK:=cmd_bIncomingDoorHandValid);

// Monitor on rising edge. The feeding machine (ie, 994-X) sets LH/RH inputs at start of its feed-out seq. 
rtrigIncomingDoorHandChanged(CLK:=cmd_bIncomingDoorHandValid AND cmd_eIncomingDoorHandLast <> cmd_eIncomingDoorHand);

cmd_eIncomingDoorHandLast := cmd_eIncomingDoorHand;

bSelectedDestinationIndexChanged := cmd_iSelectedDestinationIndexLast <> cmd_iSelectedDestinationIndex;
cmd_iSelectedDestinationIndexLast := cmd_iSelectedDestinationIndex;


bAutoDataReadyConfigChanged := bAutoDataReadyConfigLast <> config_bAutoDataReady;
bAutoDataReadyConfigLast := config_bAutoDataReady;

rtrigAutoDataReadyChanged(clk:=bAutoDataReadyConfigChanged);

IF bSelectedDestinationIndexChanged OR bAutoDataReadyConfigChanged THEN
	setDoorDataReadyLatch(FALSE);
END_IF

tofSelectedDestinationIndexChangedTimer(IN := bSelectedDestinationIndexChanged, PT := T#100MS);

// Detect falling edge of the input signal
ftrigSelectedDestinationIndexChanged(CLK := tofSelectedDestinationIndexChangedTimer.Q);

IF ftrigSelectedDestinationIndexChanged.Q THEN	
	bAnySourceDestinationIndexFeedoutPortEnabled := anySourceDestinationIndexFeedoutPortEnabled(UINT_TO_INT(cmd_iSelectedDestinationIndex));
	cmd_bRetry := config_bAutoDataReady AND bWaitingForClearRoute AND NOT bHasDoor AND bAnySourceDestinationIndexFeedoutPortEnabled;
	IF NOT bAnySourceDestinationIndexFeedoutPortEnabled THEN
		logger.fbFString(sFormat := 'Table [%s]: No feed-out ports found for the selected destination index [%d].', 
			arg1 := F_STRINGEx(MAIN.mainStateMachine.smCtrlInterface.config_stTransferTableConfig.PrimaryTable.Tables[config_iTableArrayIndex].Name), 
			arg2 := F_UINT(cmd_iSelectedDestinationIndex));	
		logger(sMessage := logger.fbFString.sOut, ePriority := LOGPRIORITY_ALERT);
	END_IF
END_IF

IF config_bAutoDataReady THEN
	// When table is configured as an input and 'hungry-mode' with destination index 0 mapped to 2 or more feed-out ports,
	// and config_bAutoDataReady is True, the physical Destination Index switch and Door Ready button are not used, cmd_bDoorDataReady is not used and always False.
	
	IF ftrigIncomingDoorHandValid.Q THEN
		setDoorDataReadyLatch(FALSE);
	ELSIF rtrigIncomingDoorHandChanged.Q OR 
		ftrigSelectedDestinationIndexChanged.Q OR
		rtrigAutoDataReadyChanged.Q THEN
		bAnySourceDestinationIndexFeedoutPortEnabled := anySourceDestinationIndexFeedoutPortEnabled(UINT_TO_INT(cmd_iSelectedDestinationIndex));
		IF cmd_bIncomingDoorHandValid AND bAnySourceDestinationIndexFeedoutPortEnabled THEN
			cmd_iSelectedDestinationIndexLatched	:= cmd_iSelectedDestinationIndex;
			cmd_eIncomingDoorHandLatched			:= cmd_eIncomingDoorHand;
			cmd_sJobNameLatched						:= cmd_sJobName;
			
			// Set cmd_bDoorDataReadyLatched = True. 
			// The feeding machine (ie 994-X) automatically clears LH and RH inputs when its feed-out seq completes.
			setDoorDataReadyLatch(TRUE); 
		ELSE
			setDoorDataReadyLatch(FALSE); 
		END_IF
		
	END_IF
ELSE
	// manual simple-rounting mode. 
	rtrigDoorDataReady(CLK:=cmd_bDoorDataReady);
	IF rtrigDoorDataReady.Q THEN
		IF NOT cmd_bDoorDataReadyLatched THEN
			cmd_iSelectedDestinationIndexLatched	:= cmd_iSelectedDestinationIndex;
			cmd_sJobNameLatched						:= cmd_sJobName;
			setDoorDataReadyLatch(TRUE);
		ELSE
			setDoorDataReadyLatch(FALSE);	
		END_IF
	END_IF
	
	IF ftrigIncomingDoorHandValid.Q THEN
		setDoorDataReadyLatch(FALSE);
	ELSIF rtrigIncomingDoorHandChanged.Q THEN
		cmd_eIncomingDoorHandLatched			:= cmd_eIncomingDoorHand;
	END_IF
END_IF

IF 	rtrigRequestNewRoute.Q OR 
	rtrigTableIndexNotExistInDoorTrackTargetPath.Q 
	THEN
	// this will filter out stDoorTrack.Target in the DestinationIndex Feedout-port popup
	cmd_bNewRouteRequested := bHasDoor;  
END_IF

bCurrentTargetFeedoutPortEnabled := currentTargetFeedoutPortEnabled();
rtrigTargetFeedoutPortsDisabled(CLK:=NOT bCurrentTargetFeedoutPortEnabled);
ftrigTargetFeedoutPortsDisabled(CLK:=NOT bCurrentTargetFeedoutPortEnabled);

bAnyCurrentTargetFeedoutPortEnabled := anyCurrentTargetFeedoutPortEnabled();
bAllCurrentTargetFeedoutPortsEnabled := allCurrentTargetFeedoutPortsEnabled();
rtrigAllCurrentTargetFeedoutPortsEnabled(CLK:=bAllCurrentTargetFeedoutPortsEnabled);
ftrigAllCurrentTargetFeedoutPortsEnabled(CLK:=bAllCurrentTargetFeedoutPortsEnabled);

bAnyDestinationIndexFeedoutPortEnabled := anyDestinationIndexFeedoutPortEnabled();
_bAllTargetFeedoutPortsDisabled := 
	bHasDoor AND 
	NOT (cmd_bNewRouteRequestedFromDoorHasNoTarget OR bAnyDestinationIndexFeedoutPortEnabled OR bAnyCurrentTargetFeedoutPortEnabled) 
	;  
rtrigAllTargetFeedoutPortsDisabled(CLK:=_bAllTargetFeedoutPortsDisabled);
ftrigAllTargetFeedoutPortsDisabled(CLK:=_bAllTargetFeedoutPortsDisabled);

_bDoorHasNoTarget := cmd_bInitialized AND bHasDoor AND (stDoorTrack.Target = -1);
rtrigDoorHasNoTarget(CLK:=_bDoorHasNoTarget);
ftrigDoorHasNoTarget(CLK:=_bDoorHasNoTarget);

IF rtrigDoorHasNoTarget.Q THEN
	cmd_bDoorHasNoTarget := TRUE;
END_IF

bRequestNewRouteComplete := machineState = TABLEMANAGER_DOOR_TRACKER_FINDPATH_REQUEST_NEW_ROUTE_COMPLETE;
bWaitingForClearRoute := machineState = TABLEMANAGER_DOOR_TRACKER_FINDPATH_WAITING_FOR_CLEAR_ROUTE;
bWaitForDataReadyOrTransferredIn := machineState = TABLEMANAGER_DOOR_TRACKER_WAIT_FOR_DATA_READY_OR_TRANSFERRED_IN;
bDoorTransferringIn := machineState = TABLEMANAGER_DOOR_TRACKER_TRANSFERRING_IN;
bRouteReadyWaitForFeedIn := machineState = TABLEMANAGER_DOOR_TRACKER_ROUTE_READY_WAIT_FOR_FEED_IN;
bDoorFeedingIn := machineState = TABLEMANAGER_DOOR_TRACKER_DOOR_FEEDING_IN;
bDoorFeedingOut  := machineState = TABLEMANAGER_DOOR_TRACKER_DOOR_FEEDING_OUT;				
bDoorInMachineIdle := machineState = TABLEMANAGER_DOOR_TRACKER_DOOR_IN_MACHINE_IDLE;
bDoorWaitingForFeedOut := machineState = TABLEMANAGER_DOOR_TRACKER_WAIT_FOR_FEED_OUT;
bWaitAllTablesReady := machineState = TABLEMANAGER_DOOR_TRACKER_WAIT_ALL_TABLES_READY;
bAllTargetFeedoutPortsDisabled  := machineState = TABLEMANAGER_DOOR_TRACKER_ALL_TARGET_FEEDOUT_PORTS_DISABLED;	
bDoorHasNoTarget := machineState = TABLEMANAGER_DOOR_TRACKER_DOOR_HAS_NO_TARGET;

rtrigDoorDataReadyLatched(CLK:=cmd_bDoorDataReadyLatched);
ftrigDoorDataReadyLatched(CLK:=cmd_bDoorDataReadyLatched);
IF rtrigDoorDataReadyLatched.Q THEN
	cmd_bReroutePending := FALSE;
END_IF
IF ftrigDoorDataReadyLatched.Q THEN
	cmd_bReroutePending := TRUE;
END_IF

bAnyTableBusy := anyTableBusy();
rtrigRerouteAllTablesWaitingTransferredOut(CLK:=cmd_bReroutePending AND NOT bAnyTableBusy);
 
IF rtrigRerouteAllTablesWaitingTransferredOut.Q THEN
	cmd_bReroutePending := FALSE;
	bAnyFeedoutTableEmptyAndReady := anyFeedoutTableEmptyAndReady();
	IF bAnyFeedoutTableEmptyAndReady THEN
		// send reroute request to all tables who were blocked by the Data Ready Latch.
		// For example, SN6 layout has 5 tables and 2 columns. 
		// T1 has Data Ready Latch active, doors on T2 or T3 cannot go to T5 when T5 became empty, then Data Ready latch is turned off.
		rerouteAllTablesWaitingTransferredOut();
	END_IF	
END_IF

bReadyToFeedout := 
	bHasDoor AND 
	stDoorTrack.Target = config_iTableArrayIndex AND 
	bAnyCurrentTargetFeedoutPortEnabled AND
	NOT (stDoorTrack.DoorRotateRequired XOR stDoorTrack.DoorWasRotated);
			
rtrigReadyToFeedout(CLK:=bReadyToFeedout);
ftrigReadyToFeedout(CLK:=bReadyToFeedout);



rtrigAnyCurrentTargetFeedoutPortEnabled(CLK:=
	bAnyCurrentTargetFeedoutPortEnabled);
ftrigAnyCurrentTargetFeedoutPortEnabled(CLK:= 	 
	bAnyCurrentTargetFeedoutPortEnabled);

rtrigAnyDestinationIndexFeedoutPortEnabled(CLK:=
 	bAnyDestinationIndexFeedoutPortEnabled);

ftrigAnyDestinationIndexFeedoutPortEnabled(CLK:=
 	bAnyDestinationIndexFeedoutPortEnabled);		
	
rtrigAnyTableDoorTrackTargetChanged(CLK:=
	pStatus_bAnyTableDoorTrackTargetChanged^
	);
IF rtrigAnyTableDoorTrackTargetChanged.Q OR 
	//rtrigAnyCurrentTargetFeedoutPortEnabled.Q OR
	//rtrigAnyDestinationIndexFeedoutPortEnabled.Q OR 
	ftrigTargetFeedoutPortsDisabled.Q OR
	rtrigDoorDataReady.Q 
	THEN
	cmd_bRetry := TRUE;
END_IF

ftrigNewRouteRequestedFromAllTargetFeedoutPortsDisabled(CLK:=cmd_bNewRouteRequestedFromAllTargetFeedoutPortsDisabled);
ftrigNewRouteRequestedFromDoorHasNoTarget(CLK:=cmd_bNewRouteRequestedFromDoorHasNoTarget);

IF downstream.status_bDownstreamError THEN
	iErrorId := TABLEMANAGER_DOWNSTREAM_ERROR;
END_IF

IF iErrorId <> 0 THEN
	raiseError(FALSE);
END_IF

IF NOT cmd_bEnable THEN
	IF machineState > TABLEMANAGER_ENABLING AND
		machineState <= TABLEMANAGER_ERROR THEN
		machineState := TABLEMANAGER_DISABLED;
	END_IF	
ELSIF bError THEN
	IF machineState > TABLEMANAGER_ENABLING AND
		machineState < TABLEMANAGER_ERROR THEN
		machineState := TABLEMANAGER_ERROR;
	END_IF	
ELSIF ftrigNewRouteRequestedFromDoorHasNoTarget.Q OR 
	cmd_bDoorHasNoTarget THEN
	IF machineState >= TABLEMANAGER_DOOR_TRACKER_START AND
		machineState < TABLEMANAGER_DOOR_TRACKER_DOOR_HAS_NO_TARGET THEN
		machineState := TABLEMANAGER_DOOR_TRACKER_DOOR_HAS_NO_TARGET;
	END_IF
ELSIF ftrigNewRouteRequestedFromAllTargetFeedoutPortsDisabled.Q OR
	rtrigAllTargetFeedoutPortsDisabled.Q THEN
	IF machineState >= TABLEMANAGER_DOOR_TRACKER_START AND
		machineState < TABLEMANAGER_DOOR_TRACKER_ALL_TARGET_FEEDOUT_PORTS_DISABLED THEN
		machineState := TABLEMANAGER_DOOR_TRACKER_ALL_TARGET_FEEDOUT_PORTS_DISABLED;
	END_IF
ELSIF NOT cmd_bAutoFeedOn THEN
	IF machineState > TABLEMANAGER_AUTOFEED_OFF AND
		machineState < TABLEMANAGER_ERROR THEN
		machineState := TABLEMANAGER_AUTOFEED_OFF;
	END_IF
END_IF
END_METHOD

METHOD raiseError
VAR_INPUT
	bSetError : BOOL;
END_VAR
CASE iErrorId OF
	TABLEMANAGER_DOWNSTREAM_ERROR: 
		formatError('Downstream error', 'Reset machine');
END_CASE
SUPER^.raiseError(bSetError);
END_METHOD

METHOD readInputs
VAR_INPUT
END_VAR
//smC234FeedManager
IF (config_pstHcTransferTableHardware <> 0) THEN
	// 00 - 07
	smC234FeedManager.di_DoorDataReady 			:= config_pstHcTransferTableHardware^.di_DoorDataReady 		;
	smC234FeedManager.di_IncomingDoorLH			:= config_pstHcTransferTableHardware^.di_IncomingDoorLH		;
	smC234FeedManager.di_IncomingDoorRH			:= config_pstHcTransferTableHardware^.di_IncomingDoorRH		;
	smC234FeedManager.di_DestinationBit0		:= config_pstHcTransferTableHardware^.di_DestinationBit0	;
	smC234FeedManager.di_DestinationBit1		:= config_pstHcTransferTableHardware^.di_DestinationBit1	;
	smC234FeedManager.di_DestinationBit2		:= config_pstHcTransferTableHardware^.di_DestinationBit2	;
	smC234FeedManager.di_InMachineEye			:= config_pstHcTransferTableHardware^.di_InMachineEye		;
	smC234FeedManager.di_DoorStop1Eye			:= config_pstHcTransferTableHardware^.di_DoorStop1Eye		;

	// 10 - 17           
	smC234FeedManager.di_DoorStop3Eye			:= config_pstHcTransferTableHardware^.di_DoorStop3Eye		;
	//di_JambKickoverEye - in SM_TableManager
	smC234FeedManager.di_ASideDoorSenseEye		:= config_pstHcTransferTableHardware^.di_DoorSenseEyeSideA	;
	smC234FeedManager.di_OkToFeedOutSideA		:= config_pstHcTransferTableHardware^.di_OkToFeedOutSideA	;
	smC234FeedManager.di_DisableFeedoutSideA	:= config_pstHcTransferTableHardware^.di_DisableFeedoutSideA;
	smC234FeedManager.di_BSideDoorSenseEye		:= config_pstHcTransferTableHardware^.di_DoorSenseEyeSideB	;
	smC234FeedManager.di_OkToFeedOutSideB		:= config_pstHcTransferTableHardware^.di_OkToFeedOutSideB	;
	smC234FeedManager.di_DisableFeedoutSideB	:= config_pstHcTransferTableHardware^.di_DisableFeedoutSideB;

	// 20 - 27           
	smC234FeedManager.di_CSideDoorFeedEye		:= config_pstHcTransferTableHardware^.di_DoorSenseEyeSideC	;
	smC234FeedManager.di_OkToFeedOutSideC		:= config_pstHcTransferTableHardware^.di_OkToFeedOutSideC	;
	smC234FeedManager.di_DisableFeedoutSideC	:= config_pstHcTransferTableHardware^.di_DisableFeedoutSideC;
	smC234FeedManager.di_DSideDoorFeedEye		:= config_pstHcTransferTableHardware^.di_DoorSenseEyeSideD	;
	smC234FeedManager.di_OkToFeedOutSideD		:= config_pstHcTransferTableHardware^.di_OkToFeedOutSideD	;
	smC234FeedManager.di_DisableFeedoutSideD	:= config_pstHcTransferTableHardware^.di_DisableFeedoutSideD;
	smC234FeedManager.di_AtFarFenceEye			:= config_pstHcTransferTableHardware^.di_AtFenceEyeSideC	; // "far" side
	smC234FeedManager.di_AtNearFenceEye			:= config_pstHcTransferTableHardware^.di_AtFenceEyeSideD	; // "near" side

// smC235FeedManager
ELSIF (config_pstHcConveyorHardware <> 0) THEN
	smC235FeedManager.di_CSideDoorFeedEye := config_pstHcConveyorHardware^.di_DoorSenseEyeSideC;
	smC235FeedManager.di_DSideDoorFeedEye := config_pstHcConveyorHardware^.di_DoorSenseEyeSideD;
END_IF
END_METHOD

(* base implementation to record state calling history. 
 	Derrived FB's should override this method to replace the machine' specific type of eState *)
	
METHOD recordStateCallHistory
VAR_INPUT
	iState				: INT;
	iSubState			: INT;
END_VAR
VAR
	sCurTaskCycle 		: STRING;
    eState       		: E_TableManager_States; // todo: replace with the derrived STRUCT type (ie, E_HeadManager_States)
    eSubState			: E_SubState;
END_VAR
// DO NOT CHANGE BELOW!!!
// This was auto-generated by a Kval's UML tool.

sCurTaskCycle := TO_STRING(mainStateCallingData[iState, iSubState].nCycleIdFirstCall);
eState := iState;
eSubState := iSubState;

// Enter the state name into array
mainStateCallHistory[iStateCallHistoryIndex].sTaskCycle := sCurTaskCycle;
mainStateCallHistory[iStateCallHistoryIndex].sStateId := TO_STRING(iState);
mainStateCallHistory[iStateCallHistoryIndex].sStateDesc := TO_STRING(eState);
mainStateCallHistory[iStateCallHistoryIndex].sSubStateId := TO_STRING(iSubState);
mainStateCallHistory[iStateCallHistoryIndex].sSubStateDesc := TO_STRING(eSubState);

iStateCallHistoryIndex := iStateCallHistoryIndex + 1;
IF iStateCallHistoryIndex = MAX_STATE_CALL_HISTORY THEN
	iStateCallHistoryIndex := 0;
END_IF

// mark next index to record state call history
mainStateCallHistory[iStateCallHistoryIndex].sTaskCycle := '--';
mainStateCallHistory[iStateCallHistoryIndex].sStateId := '--';
mainStateCallHistory[iStateCallHistoryIndex].sStateDesc := '--';
mainStateCallHistory[iStateCallHistoryIndex].sSubStateId := '--';
mainStateCallHistory[iStateCallHistoryIndex].sSubStateDesc := '--';
END_METHOD

METHOD rerouteAllTablesWaitingTransferredOut
VAR 
	i : INT;
END_VAR
FOR i:=0 TO MAIN.mainStateMachine.smCtrlInterface.config_stTransferTableConfig.PrimaryTable.TablesCount-1 DO
	IF NOT MAIN.mainStateMachine.smCtrlInterface.config_stTransferTableConfig.PrimaryTable.Tables[i].IsFunctionalTable THEN
		CONTINUE;
	END_IF
	IF (//MAIN.mainStateMachine.asmTableManagers[i].bDoorTransferringIn OR 
		MAIN.mainStateMachine.asmTableManagers[i].bDoorInMachineIdle) AND 
		
		// any of these is true, skip sending reroute.		
		NOT (//MAIN.mainStateMachine.asmTableManagers[i].status_bBusy OR
			MAIN.mainStateMachine.asmTableManagers[i].stDoorTrack.Target = i)

		THEN
		MAIN.mainStateMachine.asmTableManagers[i].cmd_bReroute := TRUE;
	END_IF
END_FOR
END_METHOD

METHOD resetDoorTrack
VAR_INPUT
END_VAR
stDoorTrack.Source := config_iTableArrayIndex;
stDoorTrack.DestinationIndex := UINT_TO_INT(cmd_iSelectedDestinationIndexLatched);
stDoorTrack.DoorHand := cmd_eIncomingDoorHandLatched;
stDoorTrack.Name := cmd_sJobNameLatched;
END_METHOD

(* Any trigger that caused state transition (ie, cmd_bHome, cmd_bStartSequence, etc..) that
 	needs to be reset should go in here.
	 
	NOTE: The derived function block of KvalStateMachineBase_UmlSC should override/extend this method. *)
METHOD resetTriggers
SUPER ^.resetTriggers();
//TODO: reset all triggers (ie, cmd_bHome, cmd_bPark, etc...) here...
END_METHOD

METHOD setDestinationIndex
VAR_INPUT
	iDestinationIndex : UINT;
END_VAR
cmd_iSelectedDestinationIndex := iDestinationIndex;
END_METHOD

METHOD setDoorDataReady
VAR_INPUT
	bDoorDataReady : BOOL;
END_VAR
cmd_bDoorDataReady := bDoorDataReady;
END_METHOD

METHOD setDoorDataReadyLatch
VAR_INPUT
	bLatched : BOOL;
END_VAR
cmd_bDoorDataReadyLatched := bLatched;
smC234FeedManager.setDoorDataAck(bLatched);
END_METHOD

METHOD setDoorTrack
VAR_INPUT
	stDoorTrackOther : ST_DoorTrack;
END_VAR
// is the target's door-dasher busy?
IF smDoorDasher.bTransferring THEN
	stDoorTrackLast := stDoorTrackOther;
	bDoorTrackDirty := TRUE;
ELSE
	stDoorTrack := stDoorTrackOther;
	setTableEmptyStatus(FALSE);
END_IF
END_METHOD

METHOD setDoorTransferredInCompleted
VAR_INPUT
END_VAR
cmd_bDoorTransferInCompleted := TRUE;
END_METHOD

METHOD setDoorTransferredInStarted
VAR_INPUT
END_VAR
cmd_bDoorTransferInStarted := TRUE;
END_METHOD

METHOD setExternal
VAR_INPUT
END_VAR
bExternal := TRUE;
smC234FeedManager.cmd_bExternal := TRUE;
smC235FeedManager.cmd_bExternal := TRUE;
END_METHOD

METHOD setFeedInStarted
VAR_INPUT
END_VAR
cmd_bFeedinStarted := TRUE;
END_METHOD

METHOD setFeedOutStarted
VAR_INPUT
END_VAR
cmd_bFeedoutStarted := TRUE;
END_METHOD

METHOD setIncomingDoorHand
VAR_INPUT
	eIncomingDoorHand					: E_DOORHAND;
END_VAR
cmd_eIncomingDoorHand := eIncomingDoorHand;
END_METHOD

METHOD setInternal
VAR_INPUT
END_VAR
smC234FeedManager.cmd_bInternal := TRUE;
smC235FeedManager.cmd_bInternal := TRUE;
END_METHOD

METHOD setJobProcessingPhase
VAR_INPUT
	eJobPhase : E_JobProcessingPhases;
END_VAR
IF config_bCanFeedinFromSideA THEN
	fbJobSync.setJobProcessingPhase(eInJpp:=eJobPhase);
END_IF
END_METHOD

METHOD setNewTargetFeedoutPortSelected
VAR_INPUT
	stDoorTrackOther : ST_DoorTrack;
END_VAR
cmd_bNewTargetFeedoutPortSelected := 
	bHasDoor
;
IF cmd_bNewTargetFeedoutPortSelected THEN
	cmd_stNewTargetFeedoutPort.TableIndex := stDoorTrackOther.Target;
	cmd_stNewTargetFeedoutPort.Side := stDoorTrackOther.TargetFeedoutSide;
END_IF
END_METHOD

METHOD setNextDoorId
VAR_INPUT	
END_VAR
VAR 
	i : INT;
	doorId : INT;
	doorIdInUsed : BOOL;
END_VAR
stDoorTrack.DoorId := 0;
FOR doorId := 1 TO MAIN.mainStateMachine.smCtrlInterface.config_stTransferTableConfig.PrimaryTable.TablesCount DO
	doorIdInUsed := FALSE;
	FOR i:=0 TO MAIN.mainStateMachine.smCtrlInterface.config_stTransferTableConfig.PrimaryTable.TablesCount-1 DO
		IF NOT MAIN.mainStateMachine.smCtrlInterface.config_stTransferTableConfig.PrimaryTable.Tables[i].IsFunctionalTable THEN
			CONTINUE;
		END_IF
		IF MAIN.mainStateMachine.asmTableManagers[i].bHasDoor AND MAIN.mainStateMachine.asmTableManagers[i].stDoorTrack.DoorId = doorId THEN
			doorIdInUsed := TRUE;
			EXIT;
		END_IF
	END_FOR
	IF NOT doorIdInUsed THEN
		stDoorTrack.DoorId := doorId;
		RETURN;
	END_IF
END_FOR
END_METHOD

METHOD setOkToFeedOutSidesTest
VAR_INPUT
END_VAR
IF config_bNoHardwareTestMode THEN
	IF config_bIsConveyorTable THEN
		smC235FeedManager.di_OkToFeedOutSideC := TRUE;
		smC235FeedManager.di_OkToFeedOutSideD := TRUE;
	ELSE
		smC234FeedManager.di_OkToFeedOutSideA := TRUE;
		smC234FeedManager.di_OkToFeedOutSideB := TRUE;
		smC234FeedManager.di_OkToFeedOutSideC := TRUE;
		smC234FeedManager.di_OkToFeedOutSideD := TRUE;
	END_IF
END_IF
END_METHOD

METHOD setReadyToFeedoutSide
VAR_INPUT
	bReadyToFeedoutSide : BOOL;
END_VAR
IF config_bIsConveyorTable THEN
	IF smC235FeedManager.cmd_eFeedoutSide = E_FeedoutSideType.C THEN
		smC235FeedManager.setReadyToFeedoutSideC(bReadyToFeedoutSide);
	ELSIF smC235FeedManager.cmd_eFeedoutSide = E_FeedoutSideType.D THEN
		smC235FeedManager.setReadyToFeedoutSideD(bReadyToFeedoutSide);
	END_IF
ELSE	
	IF smC234FeedManager.cmd_eFeedoutSide = E_FeedoutSideType.A THEN
		smC234FeedManager.setReadyToFeedoutSideA(bReadyToFeedoutSide);
	ELSIF smC234FeedManager.cmd_eFeedoutSide = E_FeedoutSideType.B THEN
		smC234FeedManager.setReadyToFeedoutSideB(bReadyToFeedoutSide);
	ELSIF smC234FeedManager.cmd_eFeedoutSide = E_FeedoutSideType.C THEN
		smC234FeedManager.setReadyToFeedoutSideC(bReadyToFeedoutSide);
	ELSIF smC234FeedManager.cmd_eFeedoutSide = E_FeedoutSideType.D THEN
		smC234FeedManager.setReadyToFeedoutSideD(bReadyToFeedoutSide);
	END_IF
END_IF
END_METHOD

METHOD setReadyToFeedoutSides
VAR_INPUT
	bReadyToFeedoutSide : BOOL;
END_VAR
smC234FeedManager.setReadyToFeedoutSideA(bReadyToFeedoutSide);
smC234FeedManager.setReadyToFeedoutSideB(bReadyToFeedoutSide);
smC234FeedManager.setReadyToFeedoutSideC(bReadyToFeedoutSide);
smC234FeedManager.setReadyToFeedoutSideD(bReadyToFeedoutSide);
smC235FeedManager.setReadyToFeedoutSideC(bReadyToFeedoutSide);
smC235FeedManager.setReadyToFeedoutSideD(bReadyToFeedoutSide);
END_METHOD

METHOD setTableEmptyStatus
VAR_INPUT
	bEmpty : BOOL;
END_VAR
IF config_bIsConveyorTable THEN
	smC235FeedManager.setTableEmptyStatus(bEmpty);
ELSE
	smC234FeedManager.setTableEmptyStatus(bEmpty);
END_IF
END_METHOD

METHOD setTablesInitialized
VAR_INPUT
	bInitialized : BOOL;
END_VAR
cmd_bInitialized := bInitialized;
END_METHOD

METHOD setTransferOutStarted
VAR_INPUT
END_VAR
IF bDoorWaitingForFeedOut THEN
	cmd_bDoorTransferOutStarted := TRUE;
ELSIF bDoorInMachineIdle THEN
	cmd_bDoorTransferOutStartedFromIdle := TRUE;
END_IF
END_METHOD

METHOD stop
VAR_INPUT
END_VAR
psmHcFeedMotor^.cmd_bStop := TRUE;
END_METHOD

(* Each transition has either or both a trigger (ie, cmd_bHome, cmd_bStartSequence, etc..)
	and a guard condition (i.e., bHeadReady AND bTableReady).
	This method updates all the state transitions.
	 
	NOTE: The derived function block of KvalStateMachineBase_UmlSC MUST override/extend this method. *)
METHOD updateStateTransitions
END_METHOD

METHOD writeOutputs
VAR_INPUT
END_VAR
//smC234FeedManager
IF (config_pstHcTransferTableHardware <> 0) THEN
	config_pstHcTransferTableHardware^.do_DoorDataAck 			:= smC234FeedManager.do_DoorDataAck			;
	config_pstHcTransferTableHardware^.do_OkToFeedInSideA		:= smC234FeedManager.do_OkToFeedInSideA		;
	config_pstHcTransferTableHardware^.do_ReadyToFeedoutSideA	:= smC234FeedManager.do_ReadyToFeedoutSideA	;
	config_pstHcTransferTableHardware^.do_ReadyToFeedoutSideB	:= smC234FeedManager.do_ReadyToFeedoutSideB	;
	config_pstHcTransferTableHardware^.do_ReadyToFeedoutSideC	:= smC234FeedManager.do_ReadyToFeedoutSideC	;
	config_pstHcTransferTableHardware^.do_ReadyToFeedoutSideD	:= smC234FeedManager.do_ReadyToFeedoutSideD	;
// smC235FeedManager - has no outputs
END_IF
END_METHOD

END_FUNCTION_BLOCK

(* stored: Version 1.1.0.1, ProductVersion 3.1.4024.14
   POU SM_TableManager: Id {174d8473-0e60-42e3-8b03-499b71e99b59}, SpecialFunc None
   Folder DoorTracker: Id {50b69c24-2b46-43e3-b36d-b1d70cbe5b58}
   Folder test: Id {0084e85f-cd3b-4f14-9299-47ac4407d6d3}
   Folder uml: Id {b233606c-76f3-41a1-888b-a52054d89419}
   Method addCandidateRouteToDoorTrack: Id {8c7f58ec-3e89-4dd4-a089-fedc2436e767}
   Method addSearchResultToDoorTrack: Id {b8af4a55-7728-432a-9950-e14343bd6d88}
   Method addToAllEnabledFeedoutPorts: Id {554e2fc3-9d5d-4d26-9e50-2f48d062c7b7}
   Method addToRejectedFeedoutPorts: Id {d5b4eb84-451f-4e54-b76e-7943fbdb78c0}
   Method addToReroutableFeedoutPorts: Id {a3b4532f-b9e9-4082-9659-e3431dedea73}
   Method addToTargetFeedoutPorts: Id {0e331e33-4cbf-43b3-9477-7af6b8f5d636}
   Method allChildrenAutoFeedOn: Id {daf1b790-c780-47ce-a169-64f8884225d5}
   Method allCurrentTargetFeedoutPortsEnabled: Id {f2006f4e-4f1d-446d-84a2-0b39c5c3a97e}
   Method allTablesReady: Id {2be8f198-4a7b-479e-8439-d0483fd5d5e1}
   Method anyChildAutofeedOn: Id {c1a08391-408e-45a6-b34d-10e5a7ada541}
   Method anyChildBusy: Id {3aa41549-7841-4207-b717-924a8b446692}
   Method anyChildExternal: Id {f97a57f3-2094-4d29-9be5-cfab42b82825}
   Method anyCurrentTargetFeedoutPortEnabled: Id {3c837b95-e21c-4e93-ae8b-779a6f9902c6}
   Method anyDestinationIndexFeedoutPortEnabled: Id {12b3bad6-2022-4e0e-a42d-a3610a5beab4}
   Method anyDoorDasherBusy: Id {0bafcac9-6d4d-4eb2-9d39-51241300d7cb}
   Method anyFeedoutTableEmptyAndReady: Id {ee556320-a2ce-4102-9eb3-715bd6daaac6}
   Method anyNeighboringTableBusy: Id {7bb14e94-bfdb-45d0-a989-283d70e92cf8}
   Method anyNeighboringTableEmpty: Id {a35b862f-9491-484d-ad97-741a63d04fef}
   Method anyNeighboringTableEmptyAndNotInPath: Id {09776181-5163-48bc-9ad2-53d2f67d6d60}
   Method anyNeighboringTableHasDoorAndDataReadyActive: Id {4bc8dfe2-fb04-4977-9f25-83269968d28e}
   Method anySourceDestinationIndexFeedoutPortEnabled: Id {9634d36c-8dae-42cf-afd4-bcabe9ec781c}
   Method anyTableBusy: Id {a539711d-fe63-485b-9b11-f284ed7380f1}
   Method anyTableEmpty: Id {162a345e-4dbd-42c2-878f-4bacdfd75dc4}
   Method anyTableWithDoorHasNoTarget: Id {e2c67dc4-33fd-4884-b9f1-f45179f63cf1}
   Method autofeedOff: Id {906806cd-13af-4bd1-b8b1-431a1fe0d2de}
   Method autofeedOn: Id {3a34afc0-a689-4d77-ab4b-85813a8d5a08}
   Method blinkReadyToFeedoutSideA: Id {40afdf22-7ce5-4ef1-a1c3-33a417624aa6}
   Method blinkReadyToFeedoutSideB: Id {c8e3469f-eb89-49cd-a018-2b81dd5481b0}
   Method blinkReadyToFeedoutSideC: Id {abff8d64-eeda-41cd-a5d1-74bc3097acb8}
   Method blinkReadyToFeedoutSideD: Id {e194fc37-7c0a-44ee-9450-4ecdfe5f3fb5}
   Method blinkReadyToFeedoutSides: Id {41d4f0b5-5c58-4523-9be3-4127591d0332}
   Method clearDoorTrack: Id {444cf8e5-655d-44ea-b81d-0e65b3dcc0d2}
   Method clearDoorTrackDoorIdAndTarget: Id {d5e1a048-836e-406f-a96c-3657c5cd3d3d}
   Method clearLastError: Id {8f780761-7cf2-4845-9ab3-b61851f020c1}
   Method clearNextDoorId: Id {6291adc0-8776-45ab-ab12-88f9fd1b75e3}
   Method computeDirectionalChanges: Id {7a81d0e5-e764-4e97-8ad2-e86baa26fc5e}
   Method computeDoorsInPath: Id {ad297419-b722-47ac-9a42-76e356776bf5}
   Method computeFinalScore: Id {75c159b4-96a0-4001-b0b0-9e9b3f8a8942}
   Method currentTargetFeedoutPortEnabled: Id {fd5f3e03-c897-44c1-8236-b5182b87fd5c}
   Method doesPathRequireRotation: Id {0b327541-31ff-4a5c-86bd-9d0f3be5970e}
   Method doState: Id {6a4cbce2-2fc3-4e59-823c-ed92f85a8b31}
   Method doState_UmlSC: Id {ca9a05d5-ef1f-4383-81e8-fa84a01166e3}
   Method existTableIndexInDoorTrackTargetPath: Id {07bb07fc-e9b4-4b09-be22-83530d508919}
   Method findAllCandidateRoutes: Id {777404d9-c9f9-4229-aa62-02f204a97067}
   Method findAllEnabledFeedoutPorts: Id {02d3a3c2-6e9d-4d52-a9fc-fd4c54c43222}
   Method findCandidateRoute: Id {5c12861c-70f7-41d8-b3df-46a2a0c2735f}
   Method findSearchResults: Id {bd51969a-c2df-4d6f-8ba6-d74e19005115}
   Method getFeedMgrStateDescription: Id {dd4f8096-e826-44c5-a4b8-964b0c5c1cdc}
   Method getSourceAndDestinationIndexFeedoutPortsCount: Id {07e1c1da-b6a8-43fe-9ff3-344650038134}
   Method getStateDescription: Id {ae6ca58b-2396-47fd-8ebe-ee8f2a4fd647}
   Method getTargetNodeDirection: Id {03a0f889-dd12-4ae3-9914-2ae956fdcf7d}
   Method goFast: Id {d15efc3d-6a96-4af5-af7a-e87f5fb70bc4}
   Method goFwd: Id {ed06c3d8-4e20-4433-850f-6812a1a5f4d0}
   Method goRev: Id {5881d02a-e7f3-4951-a9fe-2d7975530b1f}
   Method goSlow: Id {ae79a980-f8ab-4261-bbc3-f3ffc239285c}
   Method hasDeadlockedDoorInPath: Id {7d767058-f468-42fc-9c91-690e29e49ed4}
   Method hasDoorGoingOppositeDirection: Id {d03ba15b-9e9a-473e-a09b-09f80459e23b}
   Method hasEmptyTableInPath: Id {3fc6f488-6f3b-48f0-9665-4db354def7f8}
   Method hasError: Id {2c61bbda-1b42-49bc-8a59-a85cdaf154bd}
   Method hasErrorDescription: Id {1faa15b1-5213-4852-af31-65adb95f968b}
   Method hasErrorId: Id {9c82927c-e4ba-48de-956e-36421fafaa17}
   Method hasIncomingDoorInPath: Id {ad3e0b4b-e655-460d-af27-fbf5c8db8edd}
   Method initDoorTrack: Id {49c6cea8-7efe-4c11-a190-4a562681b896}
   Method initialize: Id {4805b685-66bc-4917-916b-42c030f9c476}
   Method initInputSourceAndDestinationIndexWithHighestFeedoutPortsCount: Id {5c4a8618-d381-4871-a72a-b30663d1ea99}
   Method isCurrentTargetFeedoutPortEnabled: Id {8fdb5738-35be-4b91-9480-4162dff3ade2}
   Method isCurrentTargetFeedoutPortExistInDestinationIndexFeedoutPorts: Id {9e6a027e-10ab-406b-b13c-55256f92c2b6}
   Method isFeedoutSideEnabled: Id {3e5b0684-7834-4279-a78d-91e7536d3ed5}
   Method isNeighborInTargetPath: Id {551b1681-1d03-4df0-b040-00154acda5c3}
   Method isTableIndexExistInCandidateRoutes: Id {4b981153-e66a-4065-9e51-719e2c8b119c}
   Method minDirectionalChanges: Id {f0a486d1-b229-4b7e-a500-6722e1ff6a71}
   Method minDoorsInPath: Id {2350c524-4230-4787-84a0-2e49f11a184b}
   Method minNumberOfHops: Id {186d5b37-6fed-4cd7-8288-763ea95336a5}
   Method pathHasRotateOption: Id {b461e24f-06ee-47cf-b679-d5591d468038}
   Method postProcess: Id {e52be110-5b4d-47d5-9fae-195b283f292e}
   Method preProcess: Id {1f65a54a-6f32-4b36-9e02-6acf916d497e}
   Method raiseError: Id {f5d9d67f-ab61-44a6-9451-bbf2e0261b43}
   Method readInputs: Id {92f8e551-5cc4-4394-850e-c9bc17fa3ca5}
   Method recordStateCallHistory: Id {1a6710e9-87c6-4b9f-92fa-ab90bada326b}
   Method rerouteAllTablesWaitingTransferredOut: Id {4b35eabe-6151-4122-80f5-943515c0eb02}
   Method resetDoorTrack: Id {172a9df1-dab2-4e9c-9477-cb7888ba8ea9}
   Method resetTriggers: Id {2057ce01-c973-4eda-a7a3-55f5fbd5ddd3}
   Method setDestinationIndex: Id {1213f6b9-4eea-436f-806f-174981d9f48d}
   Method setDoorDataReady: Id {bfcad898-487a-4556-af42-a3716dcf441d}
   Method setDoorDataReadyLatch: Id {eae2fcb4-a4c0-4f64-b7cc-987f86c7d37f}
   Method setDoorTrack: Id {dc11f6be-65db-4a9c-b496-5effd4aafce7}
   Method setDoorTransferredInCompleted: Id {6704b02e-7bd9-457e-b12b-5a45d974e5c1}
   Method setDoorTransferredInStarted: Id {5fe0aa52-b41d-4e3f-b2fd-5f1e1b183fbb}
   Method setExternal: Id {32025254-5fdd-4aa8-ae68-f7b79372a577}
   Method setFeedInStarted: Id {b8e7c4a3-3c30-4b88-bd76-a803de5f5530}
   Method setFeedOutStarted: Id {c8d8a26a-d690-4921-8109-000af5e8b9ef}
   Method setIncomingDoorHand: Id {4f52c99d-cb8e-45b9-bba6-a22b8c5e5798}
   Method setInternal: Id {9464a395-ad41-41ed-b2ea-c152bd0dee0c}
   Method setJobProcessingPhase: Id {b6fa90ba-9190-441b-a987-eeb852bbf66e}
   Method setNewTargetFeedoutPortSelected: Id {2d7f9ec5-2151-41fc-905a-30f627a21c01}
   Method setNextDoorId: Id {b6fcee3a-b6e4-44da-b88e-781a674e1d02}
   Method setOkToFeedOutSidesTest: Id {04f1118d-6181-406b-9983-1d152ac6c798}
   Method setReadyToFeedoutSide: Id {fc17bb31-531b-495b-b0df-a38ca8e8c6da}
   Method setReadyToFeedoutSides: Id {e81deb71-8bd3-46ff-9aaa-17c8aa940969}
   Method setTableEmptyStatus: Id {1e4f1b5f-a214-4d1c-8704-c21028119b61}
   Method setTablesInitialized: Id {f13bf1d7-4e00-495f-b6e6-693582d70737}
   Method setTransferOutStarted: Id {d69d0e1c-86e1-43fe-befa-f1e121eb9f04}
   Method stop: Id {01068671-847c-4bcd-beb3-8d990d12a811}
   Method updateStateTransitions: Id {c84cae62-a801-42e6-8383-ae8d4b0c646e}
   Method writeOutputs: Id {88c29df7-8dd2-4bc4-abbb-3520d3674425} *)
